PROGRAM PG_Time
VAR
	FAKE_TIME: GET_TIME;
	REAL_TIME: GET_TIME;
END_VAR

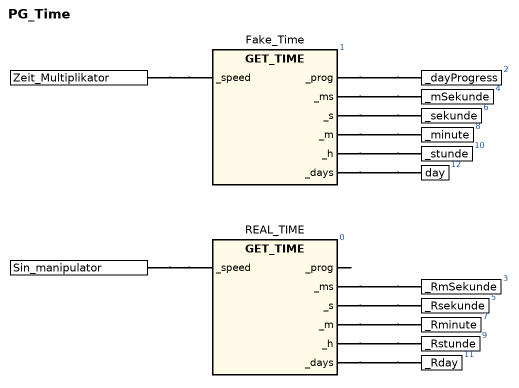
REAL_TIME(_speed := Sin_manipulator); // GET_TIME
Fake_Time(_speed := Zeit_Multiplikator); // GET_TIME
_dayProgress := Fake_Time._prog;
_RmSekunde := REAL_TIME._ms;
_mSekunde := Fake_Time._ms;
_Rsekunde := REAL_TIME._s;
_sekunde := Fake_Time._s;
_Rminute := REAL_TIME._m;
_minute := Fake_Time._m;
_Rstunde := REAL_TIME._h;
_stunde := Fake_Time._h;
_Rday := REAL_TIME._days;
day := Fake_Time._days;

END_PROGRAM

(* stored: Version 1.1.0.1, ProductVersion 3.1.4018.5
   POU PG_Time: Id {3ea9008d-fbe2-42aa-99ab-6d660e9f98ad}, SpecialFunc None *)
